// TIA Portal V17 export
// export: Created 2024-08-29T18:23:50.7159961Z, ExportSetting WithDefaults, DisplayName Totally Integrated Automation Portal, DisplayVersion V17 Update 7, DisplayName TIA Portal Openness, DisplayVersion V17 Update 7, DisplayName TIA Portal Version Control Interface, DisplayVersion V17, DisplayName SINAMICS Startdrive Advanced, DisplayVersion V17 SP2, DisplayName SINAMICS Startdrive G110M, G120, G120C, G120D, G120P, G115D, DisplayVersion V17 SP2, DisplayName SINAMICS Startdrive G130, G150, S120, S150, SINAMICS MV, S210, DisplayVersion V17 SP2, DisplayName STEP 7 Professional, DisplayVersion V17 Update 7, DisplayName STEP 7 Safety, DisplayVersion V17 Update 6, DisplayName WinCC Advanced / Unified PC, DisplayVersion V17 Update 7
VAR_GLOBAL   // PLC tag table "sequenceMemory"
   aa AT %MW1104 : Int;
   a_correctas AT %MW1100 : Int;
   a_estados AT %MW1102 : Int;
   verificacion_estados_A AT %MW1114 : Int;
   verificacion_estados_B AT %MW1116 : Int;
   b_estados AT %MW1106 : Int;
   numberOfCorrectOutputStates AT %MW1110 : Int;
   bb AT %MW1108 : Int;
   previousStep AT %MW1112 : Int;
   sequenceRestart AT %M1150.0 : Bool;
   stationTurnedOffInSequence AT %M1150.1 : Bool;
END_VAR
